ADAPTER PICKER_IN_BA (* Adapter Interface for Picker module *)
  (* Standard: 61499-1 *)
  (* Version 0.2, 2003-12-05, JHC, Rockwell Automation, Changed name from NEWADAPTER *)
  (* Version 0.1, 2002-01-08, JHC, Rockwell Automation, Added IND/RSP, renamed data, added sequences. *)
  (* Version 0.0, 2000-05-27, JHC, Rockwell Automation *)
  (* Compiler header: package fb.rt.pnp; *)
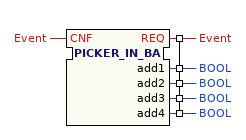
  EVENT_INPUT
    CNF; (* Confirmation from Plug *)
  END_EVENT
  EVENT_OUTPUT
    REQ WITH add1, add2, add3, add4; (* Request from Socket *)
  END_EVENT
  VAR_OUTPUT
    add1 : BOOL;
    add2 : BOOL;
    add3 : BOOL;
    add4 : BOOL;
  END_VAR
  SERVICE SOCKET/PLUG
    SEQUENCE request_confirm
      SOCKET.REQ(REQD) -> PLUG.REQ(REQD);
      PLUG.CNF(CNFD) -> SOCKET.CNF(CNFD);
    END_SEQUENCE
    SEQUENCE indication_response
      PLUG.IND(INDD) -> SOCKET.IND(INDD);
      SOCKET.RSP(RSPD) -> PLUG.RSP(RSPD);
    END_SEQUENCE
  END_SERVICE
END_ADAPTER
